ABB RAPID module: mSettings_Gripper.sys

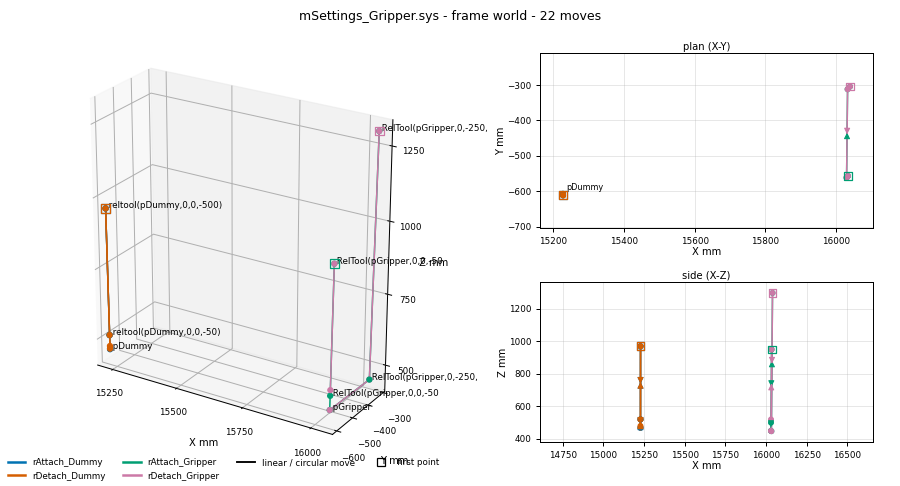
[picture p0: tool path of mSettings_Gripper.sys in frame world, 22 of 29 moves have a stored position in this frame; points joined in program order, loops and branches not executed]
MODULE mSettings_Gripper(SYSMODULE)
    !! Tools
    !! 1 geen tool
    !! 2 DUMMY
    !! 3 Grijper
    PERS num nActive_Gripper:=2;
    CONST num NoTool := 1;
    CONST num DummyTool := 2;
    CONST num GrijperTool := 3;

   !Tooldata
	PERS tooldata tGripper:=[TRUE,[[0,220.75,942],[0.5,0.5,-0.5,0.5]],[50,[0,175,400],[1,0,0,0],0,0,0]];
    ! robtargets
    CONST robtarget pDummy:=[[15227.80,-607.60,468.05],[0.00432513,-0.999965,0.00716432,0.000383958],[-1,0,-3,0],[14350,9E+09,9E+09,9E+09,9E+09,9E+09]];
    CONST robtarget pGripper:=[[16029.70,-561.83,448.04],[0.00457259,0.999965,-0.00574971,-0.00404551],[-1,-1,-3,0],[14350,9E+09,9E+09,9E+09,9E+09,9E+09]];
    !joint targets
    CONST jointtarget pHomeJoint_Grijper:=[[-10.0764,7.09903,-3.16348,0.234242,90.0265,-186.888],[14350.6,9E+09,9E+09,9E+09,9E+09,9E+09]];
    CONST jointtarget pHomeJoint_Dummy:=[[-10,-3.94306,2.59534,0.396952,1.07741,-88.065],[14350.5,9E+09,9E+09,9E+09,9E+09,9E+09]];
    !vars voor safemove
    VAR pos WZ_High_Pos;
    VAR pos WZ_Low_Pos;
    VAR shapedata WZ_Shape;
    VAR wztemporary wz_Changer_Los;

   LOCAL FUNC num fSelect_tool()
    !***************************************
    ! Func: fSelect_tool
    ! Description: manueel tool selecteren
    !***************************************
    VAR btnres nAnswer;
    CONST string Buttons_1{5}:=["Geen Tool","Dummy","Grijper","",""];
        nAnswer:=UIMessageBox(\Header:="Welke grijper tool?",\BtnArray:=Buttons_1);
        TPWrite("User selected:"+ NumToStr(nAnswer,0) + " Active:" + NumToStr(nActive_Gripper,0));
        RETURN nAnswer;
        !
   ENDFUNC

    PROC Set_Gripper_Manual()
    !***************************************
    ! Proc: Set_Gripper_Manual
    ! Description: manueel grijper actief zetten
    !***************************************
        nActive_Gripper := fSelect_tool();
        !
    ENDPROC

    PROC Get_gripper_Manual()
    !***************************************
    ! Proc: Get_gripper_Manual
    ! Description: manueel grijper wisselen
    !***************************************
     Set_Gripper(fSelect_tool());
     !
    ENDPROC


    PROC Check_gripper(num nTool)
    !***************************************
    ! Proc: Check_gripper
    ! Description: check if gripper is active
    !***************************************
        VAR btnres nAnswer;
        lbl_retry:
        IF (fGet_activeTool() <> nActive_Gripper) OR  (nActive_Gripper <> ntool) THEN
          nAnswer := UIMessageBox(\Header:="Grijper fout"\MsgArray:=["foute grijper actief !","ga manueel om grijper"],\BtnArray:=["","","","","OK"]);
          GOTO lbl_retry;
        ENDIF
        !
    ENDPROC

    PROC Check_Notool()
    !***************************************
    ! Proc: Check_Notool
    ! Description: check if too is gone
    !***************************************
        VAR btnres nAnswer;
        lbl_retry:
        CheckInput di_Changer_Tool_Aanwezig,0, \CheckTimeOut:=3,"Toolchanger sensor fout di_Changer_Tool_Aanwezig 1 ";
        !extra safety just ... because
        IF TestDI(di_Changer_Tool_Aanwezig) THEN
          nAnswer := UIMessageBox(\Header:="Grijper fout"\MsgArray:=["Tool zo los moeten zijn!","ga manueel en los op"],\BtnArray:=["","","","","OK"]);
          GOTO lbl_retry;
        ENDIF
        nActive_Gripper := NoTool;
        !
    ENDPROC

    PROC Set_Gripper(num nGripper)
    !***************************************
    ! Proc: Set_Gripper
    ! Description: get selected gripper tool
    !***************************************
        PDispOff;
        EOffsOff;
        !check if gripper io state matches selected gripper
        Check_gripper(nActive_Gripper);
        IF NOT nGripper = nActive_Gripper THEN
           go_home\Armonly;
           rDetach_tool(nActive_Gripper);
           rAttach_tool(nGripper);
           go_home\Armfirst;
        ENDIF
        Check_gripper(nGripper);
        !
    ENDPROC


    LOCAL FUNC num fGet_activeTool()
    !***************************************
    ! Func: fGet_activeTool
    ! Description: checks what tool is active
    !***************************************
    var num ntool;
        IF TestDI(di_Changer_Tool_Aanwezig)=TRUE THEN
            IF TestDI(si_Changer_Test_Grijper)=TRUE THEN
                !Grijper hangt aan de robot
                ntool:=GrijperTool;
            ELSE
                !Dummy hangt aan de robot
                ntool:=DummyTool;
            ENDIF
        ELSE
            !geen tool aan de changer of geen contact
            ntool:=NoTool;
        ENDIF
        !
    RETURN ntool;
    ENDFUNC

     LOCAL PROC rDetach_tool(num Toolnum)
    !***************************************
    ! Proc: rDetach_tool
    ! Description: drop tool on stand
    !***************************************
      TEST Toolnum
        CASE NoTool:
          !do nothing (dummy)
        CASE DummyTool:
            rDetach_Dummy;
        CASE GrijperTool:
            rDetach_Gripper;
        ENDTEST
        !
    ENDPROC

   LOCAL PROC rAttach_tool(num Toolnum)
    !***************************************
    ! Proc: rAttach_tool
    ! Description: drop tool on stand
    !***************************************
      TEST Toolnum
        CASE NoTool:
          !do nothing (dummy)
        CASE DummyTool:
            rAttach_Dummy;
        CASE GrijperTool:
            rAttach_Gripper;
        ENDTEST
        !
    ENDPROC


    LOCAL PROC rSet_Grijper_WZ()
        ! routine om wereldzones op de wisselposities te leggen
        ! in deze werledzones wordt een gesimuleerde uitgang hoog gemaakt welke in de crossconnectie om de tool te lossen gebruikt wordt
        ! buiten deze locatie kan de tool dus niet gewisseld worden in het programma
        Reset so_ChangePosition;
        WZFree wz_Changer_Los;
        IF nActive_Gripper=DummyTool THEN
            WZ_High_Pos:=[10,10,30] + pDummy.trans;
            WZ_Low_Pos:=[-10,-10,-5] + pDummy.trans;
            WZBoxDef\Inside, WZ_Shape, WZ_Low_Pos, WZ_High_Pos;
            WZDOSet\Temp,wz_Changer_Los\Inside,WZ_Shape,so_ChangePosition,1;
        ELSEIF nActive_Gripper=GrijperTool THEN
            WZ_High_Pos:=[10,10,30] + pGripper.trans;
            WZ_Low_Pos:=[-10,-10,-5] + pGripper.trans;
            WZBoxDef\Inside, WZ_Shape, WZ_Low_Pos, WZ_High_Pos;
            WZDOSet\Temp,wz_Changer_Los\Inside,WZ_Shape,so_ChangePosition,1;
        ELSE
            SET so_Changeposition;
        ENDIF
    ENDPROC

    LOCAL PROC rReset_Grijper_WZ()
       Reset so_ChangePosition;
       WZFree wz_Changer_Los;
    ENDPROC

    LOCAL PROC rAttach_Dummy()
        !
        Movej reltool(pDummy,0,0,-500),v7000,z200,tool0;
        MoveL reltool(pDummy,0,0,-50),v7000,fine,tool0;
        rToolchanger_Open;
        MoveL pDummy,v500,fine,tool0;
        !push down
        MoveL reltool(pDummy,0,0,2),v500,fine,tool0;
        rToolchanger_close \NoLockcheck;
        nActive_Gripper := DummyTool;
        Reset so_Changer_Open;
        Reset do_Gripper_Open;
        MoveL reltool(pDummy,0,0,-50),v500,fine,tool0;
        MoveL reltool(pDummy,0,0,-500),v7000,z200,tool0;
        MoveAbsJ pHomeJoint_Dummy\NoEOffs,v7000,z200,tool0;
        !
    ENDPROC

    LOCAL PROC rDetach_Dummy()
        !
        MoveAbsJ fArm_only(pHomeJoint_Dummy)\NoEOffs,v7000,z200,tool0;
        MoveAbsJ pHomeJoint_Dummy\NoEOffs,v7000,z200,tool0;
        MoveJ reltool(pDummy,0,0,-500),v7000,z200,tool0;
        MoveL reltool(pDummy,0,0,-50),v1000,z200,tool0;
        MoveL pDummy,v10,fine,tool0;
        rToolchanger_Open;
        MoveL reltool(pDummy,0,0,-10),v500,fine,tool0;
        WaitRob \InPos;
        Check_Notool;
        MoveL reltool(pDummy,0,0,-50),v500,fine,tool0;
        rReset_Grijper_WZ;
        WaitDI di_Changer_Tool_Aanwezig, 0;
        MoveL reltool(pDummy,0,0,-500),v7000,z200,tool0;
        Reset so_Changer_Open;
        !
    ENDPROC

    LOCAL PROC rAttach_Gripper()
        !
        MoveL RelTool(pGripper,0,0,-500),v7000,z200,tool0;
        MoveL RelTool(pGripper,0,0,-50),v7000,fine,tool0;
        rToolchanger_Open;
        MoveL pGripper,v50,fine,tool0;
        rToolchanger_close;
        rGripper_Open;
        nActive_Gripper := GrijperTool;
        Check_gripper(GrijperTool);
        MoveL RelTool(pGripper,0,-250,0),v500,fine,tool0;
        MoveL RelTool(pGripper,0,-250,-850),v7000,z200,tool0;
        MoveAbsJ pHomeJoint_Grijper\NoEOffs,v7000,z200,tool0;
        !
    ENDPROC


    LOCAL PROC rDetach_Gripper()
        !
        MoveAbsJ fArm_only(pHomeJoint_Grijper)\NoEOffs,v7000,z200,tool0;
        MoveAbsJ pHomeJoint_Grijper\NoEOffs,v7000,z200,tool0;
        MoveJ RelTool(pGripper,0,-250,-850),v2000,z200,tool0;
        MoveL RelTool(pGripper,0,-250,0),v1000,fine,tool0;
        MoveL pGripper,v500,fine,tool0;
        rToolchanger_Open;
        MoveL RelTool(pGripper,0,0,0-5),v50,fine,tool0;
        Check_Notool;
        MoveL RelTool(pGripper,0,0,-70),v500,fine,tool0;
        rReset_Grijper_WZ;
        MoveL RelTool(pGripper,0,0,-500),v7000,z200,tool0;
        !
    ENDPROC

    LOCAL PROC rToolchanger_Open()
    !***************************************
    ! Proc: rToolchanger_Open
    ! Description: open toolchanger
    !***************************************
      rSet_Grijper_WZ;
      Set so_Changer_Open;
      CheckInput di_Changer_Vergrendeld,0, \CheckTimeOut:=3,"Toolchanger sensor fout di_Changer_Vergrendeld 1 ";
    !
  ENDPROC

  LOCAL PROC rToolchanger_close(\switch NoLockcheck)
    !***************************************
    ! Proc: rToolchanger_close
    ! Description: sluit toolchanger
    !***************************************
      Reset so_Changer_Open;
      IF not Present(NoLockcheck) THEN
      CheckInput di_Changer_Vergrendeld,1, \CheckTimeOut:=3,"Toolchanger sensor fout di_Changer_Vergrendeld 0 ";
      endif
      CheckInput di_Changer_Tool_Aanwezig,1, \CheckTimeOut:=3,"Toolchanger sensor fout di_Changer_Tool_Aanwezig 0 ";
      rReset_Grijper_WZ;
    !
  ENDPROC

    PROC rGripper_Open()
    !***************************************
    ! Proc: rGripper_Open
    ! Description: open gripper
    !***************************************
        Reset do_Gripper_Close;
        Set do_Gripper_Open;
        !
    CheckInput si_Grijpers_Open,1, \Skip, \CheckTimeOut:=3,"Grijper sensor fout si_Grijpers_Open 0 ";
    !
  ENDPROC

    PROC rGripper_Close()
    !***************************************
    ! Proc: rGripper_Close
    ! Description: close gripper
    !***************************************
        Reset do_Gripper_Open;
        Set do_Gripper_Close;
        !
    CheckInput si_Grijpers_Dicht,1, \Skip, \CheckTimeOut:=3,"Grijper sensor fout si_Grijpers_Dicht 0 ";
    !
  ENDPROC

  FUNC bool fCheckGripperPart(\dionum  nExpection)
    !***************************************
    ! FUNC: f_checkPart
    ! Description: check if part present
    ! Handel sensor fault or ligial pos
    !***************************************
    VAR btnres nAnswer;
    VAR bool bTimeout;
    WaitRob \inpos;
    IF Present(nExpection) THEN
        WaitDI di_Sensor1_Q1_In,nExpection\MaxTime:=3\TimeFlag:=bTimeout;
        WaitDI di_Sensor2_Q1_In,nExpection\MaxTime:=3\TimeFlag:=bTimeout;
    Else
        WaitTime 2;
    ENDIF
  lbl_retry:
    IF TestDI(di_Sensor1_Q1_In) = true AND TestDi(di_Sensor2_Q1_In) = true THEN
      RETURN TRUE;
    ENDIF

    IF TestDI(di_Sensor1_Q1_In) = false AND TestDi(di_Sensor2_Q1_In) = false THEN
     RETURN FALSE;
    ENDIF

    nAnswer := UIMessageBox(\Header:="Grijper sensor fout"
    \MsgArray:=["sensoren niet zoals verwacht!","sensor di_Sensor1_Q1_In en di_Sensor1_Q2_In","moeten altijd gelijk zijn van status","corrigeer positie van balk en controleer sensoren"]
    ,\BtnArray:=["","","","","OK"]);
    GOTO lbl_retry;
    !
    ENDFUNC

   FUNC bool fCheckGripperNotInrange()
    !***************************************
    ! FUNC: fCheckGripperNotInrange
    ! Description: check if part is not  in range of sensors
    !***************************************
     WaitRob \InPos;
     WaitTime 1.5;
     IF (ai_Sensor1_Q1_in > 10) AND (ai_Sensor2_Q2_in > 2000) AND  TestDI(di_Sensor1_Q1_In) = false AND TestDI(di_Sensor2_Q1_In) = false  THEN
        RETURN TRUE;
     ENDIF
      RETURN FALSE;
    ENDFUNC

   PROC rGripper_CheckPart(bool bState \switch Supervision)
    !***************************************
    ! Proc: rGripper_CheckPart
    ! Description: check if part is present or not and part supervision
    !***************************************
    IF bState THEN
        CheckInput di_Sensor1_Q1_In,1, \Skip, \CheckTimeOut:=3,"Grijper sensor fout di_Sensor1_Q1_In";
        CheckInput di_Sensor2_Q1_In,1, \Skip, \CheckTimeOut:=3,"Grijper sensor fout di_Sensor1_Q2_In";
            IF Present(Supervision) THEN
              IDelete Int2SprvPart;
              CONNECT Int2SprvPart WITH tPartSprVsn;
              ISignalDI si_Balk_Gevonden,1,Int2SprvPart;
              IWatch Int2SprvPart;
            ENDIF
    ELSE
        CheckInput di_Sensor1_Q1_In,0, \Skip, \CheckTimeOut:=3,"Grijper sensor fout di_Sensor1_Q1_In";
        CheckInput di_Sensor2_Q1_In,0, \Skip, \CheckTimeOut:=3,"Grijper sensor fout di_Sensor1_Q2_In";
    ENDIF
    !
  ENDPROC

  PROC rGripper_PartSupervisionOff()
    !***************************************
    ! Proc: rGripper_PartSupervisionOff
    ! Description: turns off part supervision
    !***************************************
    ISleep Int2SprvPart;
    !
  ENDPROC

  TRAP tPartSprVsn
    !***************************************
    ! Trap: tPartSprVsn
    ! Description: Supervision trap that
    ! stops robot with alarm message
    ! Connected in rGripper_CheckPart
    !***************************************
   VAR btnres nAnswer;
   ISleep Int2SprvPart;
   StopMove;
   StorePath;
   nAnswer := UIMessageBox(\Header:="Grijperfout"\MsgArray:=["stuk onverwachts uit grijper","controleer de positie van het stuk in de grijper"],\BtnArray:=["","","","","Reset"]);
   RestoPath;
   IWatch Int2SprvPart;
   StartMove;
   rWait_Spindel;
  ENDTRAP

ENDMODULE
